TYPE ST_TxHmiStewart :
STRUCT
	status : DINT := 0;
	eta : ARRAY [0..5] OF REAL;
	etaRef : ARRAY [0..5] OF REAL;
	cyl : ARRAY [0..5] OF REAL;
END_STRUCT
END_TYPE

(* stored: Version 1.1.0.1, ProductVersion 3.1.4022.18
   DUT ST_TxHmiStewart: Id {a97cdde8-9053-4a79-afcc-923bad4b3e3d} *)
